{attribute addProperty BoxType "EM7004-0000-9996"}
{attribute addProperty Id "InputAT %I*ARRAY[0 ..15] OF BOOL128160"}
{attribute addProperty CRC "1547216551"}
{attribute addProperty SizeInBites "128"}
{attribute addProperty SizeInBytes "16"}
TYPE DI_Inputs_42B6F5B2 :
STRUCT
	{attribute addProperty Name "Input"}
	Input AT %I* : ARRAY[0 ..15] OF BOOL;
END_STRUCT
END_TYPE

(* stored: Version 1.2.0.0, ProductVersion 3.1.4024.9
   DUT DI_Inputs_42B6F5B2: Id {038db3a9-cf41-4e27-a934-f7fc0a37349f} *)
